PROGRAM MAIN_Burner
VAR
	State: INT;
	Delay : TON;
	IN: BOOL := TRUE;
	PT: TIME := T#5S;
	Q: INT;
	
END_VAR

IF GVL_Kitchen.System_Start = 0 THEN
 	 	Delay();
ELSE	
		CASE State OF
		0: 
		IF GVL_kitchen.Food_Spiced >0 THEN
			
			 	Delay();
			Delay(IN:=FALSE);
			GVL_kitchen.Food_Spiced := GVL_kitchen.Food_Spiced-1;
			GVL_Kitchen.Food_Cooked := GVL_Kitchen.Food_Cooked +1;
			State := 1;
			END_IF;
			
		1: 
		IF GVL_kitchen.Food_cooked > 0 THEN
				 	Delay();
			GVL_Kitchen.Food_Cooked := GVL_Kitchen.Food_Cooked -1;
			GVL_Kitchen.Food_Plated := GVL_Kitchen.Food_Plated +1;
			ELSE 
				state := 0;
			END_IF;
		END_CASE 
END_IF

END_PROGRAM

(* stored: Version 1.1.0.1, ProductVersion 3.1.4024.15
   POU MAIN_Burner: Id {f5fc2f05-488a-44f2-8202-36e07a31bae0}, SpecialFunc None *)
